// TIA Portal V19 export
TYPE "LEXCHANGETRAY_typeSR1000ControlNodeCommands"
// completionClearControlBits: LEXCHANGETRAY_typeSr1000ProfinetTelegram_completionClearControlBits
// latchandErrorClearControlBits: LEXCHANGETRAY_typeSr1000ProfinetTelegram_latchandErrorClearControlBits
// operationinstructionControlBits: LEXCHANGETRAY_typeSr1000ProfinetTelegram_operationinstructionControlBits
// parameterBankNumber: LEXCHANGETRAY_typeSr1000ProfinetTelegram_parameterBankNumber
// userData128Byte: LEXCHANGETRAY_typeSr1000ProfinetTelegram_userData128Byte
// start: Bool
// reset: Bool
// stored: Access Published
   STRUCT
      completionClearControlBits : "LEXCHANGETRAY_typeSr1000ProfinetTelegram_completionClearControlBits";
      latchandErrorClearControlBits { S7_SetPoint := 'True'} : "LEXCHANGETRAY_typeSr1000ProfinetTelegram_latchandErrorClearControlBits";
      operationinstructionControlBits { S7_SetPoint := 'True'} : "LEXCHANGETRAY_typeSr1000ProfinetTelegram_operationinstructionControlBits";
      parameterBankNumber { S7_SetPoint := 'True'} : "LEXCHANGETRAY_typeSr1000ProfinetTelegram_parameterBankNumber";
      userData128Byte { S7_SetPoint := 'True'} : "LEXCHANGETRAY_typeSr1000ProfinetTelegram_userData128Byte";
      start { S7_SetPoint := 'True'} : Bool;
      reset { S7_SetPoint := 'True'} : Bool;
   END_STRUCT;
END_TYPE
